// SIMATIC S7-200 project (STEP 7-Micro/WIN), CPU 224 REL 01.22

SYMBOL_TABLE USR1
泵2号本地启动          M1.3
泵2号远程启动          M1.2
泵1号本地启动          M1.1
泵1号远程启动          M1.0
水泵1号_启动          Q2.0
水泵1号启动           I0.0
水泵1号停止           I0.1
水泵2号启动           I0.2
水泵2号停止           I0.3
水泵3号启动           I0.4
水泵3号停止           I0.5
水泵4号启动           I0.6
水泵4号停止           I0.7
水箱加热水泵启动         I1.0
水箱加热水泵停止         I1.1
水箱加药泵启动          I1.2
水箱加药泵停止          I1.3
水泵1号启动本地         I1.4
水泵1号停止本地         I1.5
水泵2号启动本地         I2.0
水泵2号停止本地         I2.1
水泵3号启动本地         I2.2
水泵3号停止本地         I2.3
水泵4号启动本地         I2.4
水泵4号停止本地         I2.5
加水泵启动本地          I2.6
加水泵停止本地          I2.7
加药泵启动本地          I3.0
加药泵停止本地          I3.1
水泵1号泵本地          I3.2
水泵2号泵本地          I3.3
水泵3号泵本地          I3.4
水泵4号泵本地          I3.5
加水泵本地            I3.6
加药泵本地            I3.7
水泵1号过热           I4.0
水泵2号过热           I4.1
水泵3号过热           I4.2
水泵4号过热           I4.3
加水泵过热            I4.4
加药泵过热            I4.5
水箱液面低            I4.6
水泵1号启动_按钮灯       Q0.0
水泵2号启动_按钮灯       Q0.1
水泵3号启动_按钮灯       Q0.2
水泵4号启动_按钮灯       Q0.3
加水泵启动_按钮灯        Q0.4
加药泵启动_按钮灯        Q0.5
水泵1号启动_钮灯本地      Q0.6
水泵2号启动_钮灯本地      Q0.7
水泵3号启动_钮灯本地      Q1.0
水泵4号启动_钮灯本地      Q1.1
水泵2号_启动          Q2.1
水泵3号_启动          Q2.2
水泵4号_启动          Q2.3
加水泵_启动           Q2.4
加药泵_启动           Q2.5
加水泵启动_钮灯本地       Q3.0
加药泵启动_钮灯本地       Q3.1
水箱液位低            Q3.2
END_SYMBOL_TABLE

ORGANIZATION_BLOCK MAIN:OB1
TITLE=S7-200水处理程序
// [中国PLC网]http://www.cniplc.com
// 中国PLC网，中国权威PLC资讯平台，培养优秀PLC工程师！
// 本站所有例程均来自于网络，仅用于学习用途，请勿直接用于工程项目，否则产生的一切后果自负！
// 系统通过四台水泵（水泵1号启动至水泵4号启动）、一台加水泵（加水泵启动）和一台加药泵（加药泵启动）实现这些功能，确保污水处理过程高效且安全。
// 操作员既可以通过远程控制室内的按钮（如水泵1号远程启动按钮和水泵1号远程停止按钮），也可以在现场使用本地按钮（如水泵1号本地启动按钮和水泵1号本地停止按钮）及开关（如水泵1号本地开关）操作设备。
// 
// 
// 在污水处理厂的日常运行中，操作员按下水泵1号远程启动按钮时，系统首先检查水泵1号本地开关是否未启用本地模式，以及水泵1号过热传感器是否未检测到过热。
// 只有满足这些条件，水泵1号远程启动标志才会置位。
// 若水泵2号远程启动标志置位且水箱液位低传感器未检测到低液位，水泵2号启动被激活；
// 此外，水泵3、4好的远程启动逻辑也类似，若水泵3号远程启动标志置位且水箱液位低传感器未检测到低液位，水泵3号启动被激活；
// 若水泵4号远程启动标志置位且水箱液位低传感器未检测到低液位，水泵4号启动被激活。
// 随后，若水箱液位低传感器未检测到低液位，水泵1号启动被激活，同时点亮水泵1号远程启动按钮灯，提示远程控制已生效。
// 类似地，本地控制通过水泵1号本地启动按钮触发，但远程和本地控制互斥，水泵1号启动只能由其中一种方式激活。
// 水泵2号至水泵4号的控制逻辑相同，分别通过各自的按钮和传感器实现独立运行。
// 
// 
// 为了维持水箱液位，加水泵通过加水泵远程启动按钮或加水泵本地启动按钮启动。
// 然而，只有在加水泵过热传感器未检测到过热时，加水泵启动才能激活，同时点亮加水泵远程启动按钮灯或加水泵本地启动按钮灯。
// 加药泵的运行类似，通过加药泵远程启动按钮或加药泵本地启动按钮控制加药泵启动，并在加药泵过热传感器未检测到过热时生效。
// 这些设计确保加水和加药过程不会因设备故障而中断。
// 
// 系统运行时，水箱液位低传感器持续监控水箱状态。
// 若检测到低液位，水箱液位低指示灯亮起，所有泵（如水泵1号启动至加药泵启动）必须立即停止，以防止泵空转损坏设备。
// 同时，各泵的过热传感器（如水泵1号过热传感器至加药泵过热传感器）实时检测温度，一旦发现过热，相关泵的启动信号（如水泵1号远程启动标志）会复位，停止运行并保护设备。
// 例如，按下水泵1号远程停止按钮或检测到水泵1号过热传感器信号时，水泵1号启动立即关闭。
// 
// 
// 
BEGIN
Network 1 // 1#水泵远程控制
// 网络注释 
LD     水泵1号启动:I0.0
O      泵1号远程启动:M1.0
A      水泵1号停止:I0.1
A      水泵1号泵本地:I3.2
AN     水泵1号过热:I4.0
=      泵1号远程启动:M1.0
Network 2 // 1#水泵本地控制
LD     水泵1号启动本地:I1.4
LDN    水泵1号泵本地:I3.2
A      泵1号本地启动:M1.1
OLD
A      水泵1号停止本地:I1.5
AN     水泵1号过热:I4.0
=      泵1号本地启动:M1.1
Network 3 // 1#泵启动和灯
LD     泵1号远程启动:M1.0
AN     泵1号本地启动:M1.1
LD     泵1号本地启动:M1.1
AN     泵1号远程启动:M1.0
OLD
AN     水箱液面低:I4.6
=      水泵1号_启动:Q2.0
=      水泵1号启动_按钮灯:Q0.0
=      水泵1号启动_钮灯本地:Q0.6
Network 4 // 2#水泵远程控制
// 网络注释
LD     水泵2号启动:I0.2
O      泵2号远程启动:M1.2
A      水泵2号停止:I0.3
A      水泵2号泵本地:I3.3
AN     水泵2号过热:I4.1
=      泵2号远程启动:M1.2
Network 5 // 2#水泵本地控制
LD     水泵2号启动本地:I2.0
LDN    水泵2号泵本地:I3.3
A      泵2号本地启动:M1.3
OLD
A      水泵2号停止本地:I2.1
AN     水泵2号过热:I4.1
=      泵2号本地启动:M1.3
Network 6 // 2#泵启动和灯
LD     泵2号远程启动:M1.2
AN     泵2号本地启动:M1.3
LD     泵2号本地启动:M1.3
AN     泵2号远程启动:M1.2
OLD
AN     水箱液面低:I4.6
=      水泵2号_启动:Q2.1
=      水泵2号启动_按钮灯:Q0.1
=      水泵2号启动_钮灯本地:Q0.7
Network 7 // 3#水泵远程控制
// 网络注释
LD     水泵3号启动:I0.4
O      M1.4
A      水泵3号停止:I0.5
A      水泵3号泵本地:I3.4
AN     水泵3号过热:I4.2
=      M1.4
Network 8 // 3#水泵本地控制
LD     水泵3号启动本地:I2.2
LDN    水泵3号泵本地:I3.4
A      M1.5
OLD
A      水泵3号停止本地:I2.3
AN     水泵3号过热:I4.2
=      M1.5
Network 9 // 3#泵启动和灯
LD     M1.4
AN     M1.5
LD     M1.5
AN     M1.4
OLD
AN     水箱液面低:I4.6
=      水泵3号_启动:Q2.2
=      水泵3号启动_按钮灯:Q0.2
=      水泵3号启动_钮灯本地:Q1.0
Network 10 // 4#水泵远程控制
// 网络注释
LD     水泵4号启动:I0.6
O      M1.6
A      水泵4号停止:I0.7
A      水泵4号泵本地:I3.5
AN     水泵4号过热:I4.3
=      M1.6
Network 11 // 4#水泵本地控制
LD     水泵4号启动本地:I2.4
LDN    水泵4号泵本地:I3.5
A      M1.7
OLD
A      水泵4号停止本地:I2.5
AN     水泵4号过热:I4.3
=      M1.7
Network 12 // 4#泵启动和灯
LD     M1.6
AN     M1.7
LD     M1.7
AN     M1.6
OLD
AN     水箱液面低:I4.6
=      水泵4号_启动:Q2.3
=      水泵4号启动_按钮灯:Q0.3
=      水泵4号启动_钮灯本地:Q1.1
Network 13 // 加水泵远程控制
// 网络注释
LD     水箱加热水泵启动:I1.0
O      M2.0
A      水箱加热水泵停止:I1.1
A      加水泵本地:I3.6
A      加水泵过热:I4.4
=      M2.0
Network 14 // 加水泵本地控制
LD     加水泵启动本地:I2.6
LDN    加水泵本地:I3.6
A      M2.1
OLD
A      加水泵停止本地:I2.7
A      加水泵过热:I4.4
=      M2.1
Network 15 // 加水泵启动和灯
LD     M2.0
AN     M2.1
LD     M2.1
AN     M2.0
OLD
=      加水泵_启动:Q2.4
=      加水泵启动_按钮灯:Q0.4
=      加水泵启动_钮灯本地:Q3.0
Network 16 // 加药泵远程控制
// 网络注释
LD     水箱加药泵启动:I1.2
O      M2.2
A      水箱加药泵停止:I1.3
A      加药泵本地:I3.7
A      加药泵过热:I4.5
=      M2.2
Network 17 // 加药泵本地控制
LD     加药泵启动本地:I3.0
LDN    加药泵本地:I3.7
A      M2.3
OLD
A      加药泵停止本地:I3.1
A      加药泵过热:I4.5
=      M2.3
Network 18 // 加药泵启动和灯
LD     M2.2
AN     M2.3
LD     M2.3
AN     M2.2
OLD
AN     水箱液面低:I4.6
=      加药泵_启动:Q2.5
=      加药泵启动_按钮灯:Q0.5
=      加药泵启动_钮灯本地:Q3.1
Network 19
LD     水箱液面低:I4.6
=      水箱液位低:Q3.2
END_ORGANIZATION_BLOCK
